{attribute 'GeneratedUsingTerminal: EL3064-0000-0020'}
{attribute addProperty BoxType "EL3064-0000-0020"}
{attribute addProperty Id "UnderrangeBOOL1OverrangeBOOL1Limit_1BYTE1Limit_2BYTE1ErrorBOOL1TxPDO_StateBOOL1TxPDO_ToggleBOOL1"}
{attribute addProperty CRC "4073614737"}
{attribute addProperty Size "7"}
TYPE Status_F2CE6D91 :
STRUCT
	{attribute addProperty Name "Underrange"}
	Underrange : BOOL;
	{attribute addProperty Name "Overrange"}
	Overrange : BOOL;
	{attribute addProperty Name "Limit_1"}
	Limit_1 : BYTE;
	{attribute addProperty Name "Limit_2"}
	Limit_2 : BYTE;
	{attribute addProperty Name "Error"}
	Error : BOOL;
	{attribute addProperty Name "TxPDO_State"}
	TxPDO_State : BOOL;
	{attribute addProperty Name "TxPDO_Toggle"}
	TxPDO_Toggle : BOOL;
END_STRUCT
END_TYPE

(* stored: Version 1.2.0.0, ProductVersion 3.1.4024.9
   DUT Status_F2CE6D91: Id {85df2b27-182e-441e-9e55-5b2eed328319} *)
